// TIA Portal V16 export
// export: Created 2023-08-28T09:37:49.710813Z, ExportSetting WithDefaults, DisplayName Totally Integrated Automation Portal, DisplayVersion V16 Update 6, DisplayName TIA Portal Version Control Interface, DisplayVersion V16 Update 2, DisplayName TIA Portal Openness, DisplayVersion V16 Update 6, DisplayName STEP 7 Professional, DisplayVersion V16 Update 6, DisplayName STEP 7 Safety, DisplayVersion V16, DisplayName WinCC Advanced, DisplayVersion V16 Update 6
DATA_BLOCK "filtr _kalmana_2_DB_1"   // DB128
VERSION : 0.1
// stored: AutoNumber true, DBAccessibleFromOPCUA true, InstanceOfName filtr _kalmana_2, InstanceOfType FB
"filtr _kalmana_2"
BEGIN
END_DATA_BLOCK
